(* IEC 61131-3 sources: LPWCC/src, 9 files *)

(* ---- GVL.st ---- *)
VAR_GLOBAL
	IX0_0 AT %IX0.0:BOOL;
	IX0_1 AT %IX0.1:BOOL;
	IX0_2 AT %IX0.2: BOOL;
	IX0_3 AT %IX0.3: BOOL;
	IX0_4 AT %IX0.4: BOOL;
	IX0_5 AT %IX0.5: BOOL;
	IX0_6 AT %IX0.6: BOOL;
	IX0_7 AT %IX0.7: BOOL;
	IX0_8 AT %IX0.8: BOOL;

	IW6 AT %IW6:WORD;
	IW7 AT %IW7:WORD;
	IW8 AT %IW8:WORD;
	IW9 AT %IW9:WORD;
	IW10 AT %IW10:WORD;
	IW11 AT %IW11:WORD;
	IW12 AT %IW12:WORD;
	IW13 AT %IW13:WORD;

	QX0_4 AT %QX0.4:BOOL;
	QX0_5 AT %QX0.5:BOOL;
	QX0_6 AT %QX0.6:BOOL;
	QX0_7 AT %QX0.7:BOOL;
	QX1_0 AT %QX1.0:BOOL;
	QX1_1 AT %QX1.1:BOOL;
	QX3_0 AT %QX3.0:BOOL;
	QX3_1 AT %QX3.1:BOOL;
	QX3_2 AT %QX3.2:BOOL;
	QX3_3 AT %QX3.3:BOOL;
	QX3_4 AT %QX3.4:BOOL;
	QX3_5 AT %QX3.5:BOOL;
	QX3_6 AT %QX3.6:BOOL;
	QX3_7 AT %QX3.7:BOOL;
	QX4_0 AT %QX4.0:BOOL;
	QX4_1 AT %QX4.1:BOOL;
	QX4_2 AT %QX4.2:BOOL;
	QX4_3 AT %QX4.3:BOOL;
	QX4_4 AT %QX4.4:BOOL;
	QX4_5 AT %QX4.5:BOOL;
	QX4_6 AT %QX4.6:BOOL;
	QX4_7 AT %QX4.7:BOOL;
	QX5_0 AT %QX5.0:BOOL;
	QX5_1 AT %QX5.1:BOOL;
	QX5_2 AT %QX5.2:BOOL;
	QX5_3 AT %QX5.3:BOOL;
	QX5_5 AT %QX5.5:BOOL;
	QW7 AT %QW7:WORD;
	QW8 AT %QW8:WORD;
	QW9 AT %QW9:WORD;
	QW10 AT %QW10:WORD;

	ExtRestart_State:BOOL;

	TON0_M_State:BOOL;
	TON1_M_State:BOOL;
	TON2_M_State:BOOL;
	TON3_M_State:BOOL;
	TON0_A_State:BOOL;
	TON1_A_State:BOOL;
	TON2_A_State:BOOL;
	TON3_A_State:BOOL;
	TON4_A_State:BOOL;
	TON5_A_State:BOOL;
	TON6_A_State:BOOL;
	TON7_A_State:BOOL;
	TON7_1_A_State:BOOL;
	TON7_2_A_State:BOOL;
	TON8_A_State:BOOL;
	TON8_1_A_State:BOOL;
	TON8_2_A_State:BOOL;
	TON9_A_State:BOOL;
	TON10_A_State:BOOL;
	TON11_A_State:BOOL;
	TON11_1_A_State:BOOL;
	TON12_A_State:BOOL;
	TON12_1_A_State:BOOL;
	TON13_State:BOOL;
	TON14_State:BOOL;
	TON15_State:BOOL;
	TON16_Emergency_stop:BOOL;
	TON17_State:BOOL;
	TON17_SW:BOOL;
	TON18_State:BOOL;
	TON18_SW:BOOL;
	TON19_State:BOOL;
	TON20_Emergency_stop:BOOL;
	TON21_A_State:BOOL;
	TON22_A_State:BOOL;

	CAN_SET_ArcOn:BOOL;
	CAN_SET_RobotReady:BOOL;
	CAN_SET_OperMode_0:BOOL;
	CAN_SET_OperMode_1:BOOL;
	CAN_SET_OperMode_2:BOOL;
	CAN_SET_AnalogSwap:BOOL;
	CAN_SET_ProtocolMode:BOOL;
	CAN_SET_GasTest:BOOL;
	CAN_SET_WireInching:BOOL;
	CAN_SET_WireRetract:BOOL;
	CAN_SET_SourceErrReset:BOOL;
	CAN_SET_TouchSensing:BOOL;
	CAN_SET_BlowTrough:BOOL;
	CAN_SET_JOB_0:BOOL;
	CAN_SET_JOB_1:BOOL;
	CAN_SET_JOB_2:BOOL;
	CAN_SET_JOB_3:BOOL;
	CAN_SET_JOB_4:BOOL;
	CAN_SET_JOB_5:BOOL;
	CAN_SET_JOB_6:BOOL;
	CAN_SET_JOB_7:BOOL;
	CAN_SET_WeldSim:BOOL;
	CAN_SET_AnalogSetDis_0:BOOL;
	CAN_SET_AnalogSetDis_1:BOOL;
	CAN_SET_AnalogSetDis_2:BOOL;
	CAN_SET_AnalogSetDis_3:BOOL;
	CAN_SET_AnalogSetDis_4:BOOL;
	CAN_SET_AnalogSetDis_5:BOOL;
	CAN_SET_DC_AC_Disable:BOOL;
	CAN_SET_PLS_Disable:BOOL;
	CAN_SET_DC_AC:BOOL;
	CAN_SET_PLS:BOOL;
	CAN_SET_PilotArc:BOOL;

	CAN_SET_WeldCurrent:UINT;
	CAN_SET_WireHighSpd:UINT;
	CAN_SET_PLS_Ratio:UINT;
	CAN_SET_WireLowSpd:UINT;
	CAN_SET_PlasmaGasFlow:UINT;
	CAN_SET_ShieldGasFlow:UINT;

	CAN_GET_CurrFlow:BOOL;
	CAN_GET_ProcActive:BOOL;
	CAN_GET_MainCurrent:BOOL;
	CAN_GET_CollisProtect:BOOL;
	CAN_GET_PowSourReady:BOOL;
	CAN_GET_Commun_Ready:BOOL;
	CAN_GET_ErrNumber_0:BOOL;
	CAN_GET_ErrNumber_1:BOOL;
	CAN_GET_ErrNumber_2:BOOL;
	CAN_GET_ErrNumber_3:BOOL;
	CAN_GET_ErrNumber_4:BOOL;
	CAN_GET_ErrNumber_5:BOOL;
	CAN_GET_ErrNumber_6:BOOL;
	CAN_GET_ErrNumber_7:BOOL;
	CAN_GET_PLS_Sync:BOOL;
	CAN_GET_PilotArc:BOOL;
	CAN_GET_StikingRem:BOOL;
	CAN_GET_WireAvailale:BOOL;

	CAN_GET_WeldVoltage:UINT;
	CAN_GET_WeldCurrent:UINT;
	CAN_GET_MotorCurrent:UINT;
	CAN_GET_WireFeedSPD:UINT;
	CAN_GET_PlasmaGasFlw:UINT;
	CAN_GET_ShieldGasFlw:UINT;

	MW110 AT %MW110:WORD;
	MW112 AT %MW112:WORD;
	MW114 AT %MW114:WORD;
	MW116 AT %MW116:WORD;
	MW118 AT %MW118:WORD;
	MW120 AT %MW120:WORD;
	MW122 AT %MW122:WORD;
	MW124 AT %MW124:WORD;
	MW126 AT %MW126:WORD;
	MW128 AT %MW128:WORD;

	TON0_FESTO:TON;
	TON0_FESTO_STATE:BOOL;
	TON0_FESTO_SW:BOOL;
	TON1_FESTO:TON;
	TON1_FESTO_STATE:BOOL;
	TON1_FESTO_SW:BOOL;
END_VAR

VAR_GLOBAL RETAIN
	MW0 AT %MW0:WORD;
	MW2 AT %MW2:WORD;
	MW4 AT %MW4:WORD;
	MW6 AT %MW6:WORD;
	MW8 AT %MW8:WORD;
	MW10 AT %MW10:WORD;
	MW12 AT %MW12:WORD;
	MW14 AT %MW14:WORD;
	MW16 AT %MW16:WORD;
	MW18 AT %MW18:WORD;
	MW20 AT %MW20:WORD;
	MW22 AT %MW22:WORD;
	MW24 AT %MW24:WORD;
	MW26 AT %MW26:WORD;
	MW28 AT %MW28:WORD;
	MW30 AT %MW30:WORD;
	MW32 AT %MW32:WORD;
	MW34 AT %MW34:WORD;
	MW36 AT %MW36:WORD;
	MW38 AT %MW38:WORD;
	MW40 AT %MW40:WORD;
	MW44 AT %MW44:WORD;
	MW42 AT %MW42:WORD;
	MW46 AT %MW46:WORD;
	MW48 AT %MW48:WORD;
	MW50 AT %MW50:WORD;
	MW52 AT %MW52:WORD;
	MW54 AT %MW54:WORD;
	MW56 AT %MW56:WORD;
	MW58 AT %MW58:WORD;
	MW60 AT %MW60:WORD;
	MW62 AT %MW62:WORD;
	MW64 AT %MW64:WORD;
	MW66 AT %MW66:WORD;
	MW68 AT %MW68:WORD;
	MW70 AT %MW70:WORD;
	MW72 AT %MW72:WORD;
	MW74 AT %MW74:WORD;
	MW76 AT %MW76:WORD;
	MW78 AT %MW78:WORD;
	MW80 AT %MW80:WORD;
	MW82 AT %MW82:WORD;
	MW84 AT %MW84:WORD;
	MW86 AT %MW86:WORD;
	MW88 AT %MW88:WORD;
	MW90 AT %MW90:WORD;
	MW92 AT %MW92:WORD;
	MW94 AT %MW94:WORD;
	MW96 AT %MW96:WORD;
	MW98 AT %MW98:WORD;
	MW100 AT %MW100:WORD;
	MW102 AT %MW102:WORD;
	MW104 AT %MW104:WORD;

	MW130 AT %MW130:WORD;
	MW132 AT %MW132:WORD;
	MW134 AT %MW134:WORD;
	MW136 AT %MW136:WORD;
	MW138 AT %MW138:WORD;
	MW140 AT %MW140:WORD;

	MD222 AT %MD222:DWORD;
	MD232 AT %MD232:DWORD;
	MD254 AT %MD254:DWORD;
	MD304 AT %MD304:DWORD;

END_VAR

(* ---- Alarms_auto.st ---- *)
VAR
	TON13: TON;
	TON14: TON;
	TON15: TON;
	TON16: TON;
END_VAR

//Затримка аналізу аварій
TON13(IN:= MW34.10, PT:= WORD_TO_TIME(MW96), Q=> TON13_State);
//Затримка аналізу чергової дуги
TON14(IN:= TON1_A_State, PT:= WORD_TO_TIME(MW60), Q=> TON14_State);
//Затримка аналізу основної дуги
TON15(IN:= (MW34.2 AND NOT(MW34.1) AND QX5_5) OR (MW34.1 AND CAN_SET_ArcOn) OR (MW34.9 AND QX5_3), PT:= WORD_TO_TIME(MW64), Q=> TON15_State);
//Аларми
IF TON13_State THEN
	IF IX0_0 THEN MW100:= 1; MW8.1:= TRUE; END_IF //Аларм по грибку
	IF MW18.12 AND IX0_8 THEN MW100:= 2; MW8.1:= TRUE; END_IF //Аларм по аварії лазера
	IF MW18.13 AND MW34.4 AND NOT(IX0_4) THEN MW100:= 3; MW8.1:= TRUE; END_IF //Аларм по неготовності робота
	IF MW18.14 AND MW34.4 AND IX0_6 THEN MW100:= 4; MW8.1:= TRUE; END_IF //Аларм по аварії робота
	IF MW8.6 AND IW6 < MW80 THEN MW100:= 5; MW8.1:= TRUE; END_IF //Аларм по низькому тиску газу зварювання
	IF MW8.7 AND IW7 < MW82 THEN MW100:= 6; MW8.1:= TRUE; END_IF //Аларм по низькому тиску газу різання
	IF MW8.8 AND IW8 < MW84 THEN MW100:= 7; MW8.1:= TRUE; END_IF //Аларм по низьких витратах газу зварювання
	IF MW8.9 AND IW9 < MW86 THEN MW100:= 8; MW8.1:= TRUE; END_IF //Аларм по низьких витратах газу різання
END_IF
IF MW8.12 AND MW18.8 AND TON13_State AND QX5_5 AND IW12 < MW92 THEN MW100:= 9; MW8.1:= TRUE; END_IF //Аларм по низькому струму різання
IF MW8.13 AND MW18.8 AND TON13_State AND QX5_5 AND IW13 < MW94 THEN MW100:= 10; MW8.1:= TRUE; END_IF //Аларм по низькій напрузі різання
IF MW8.10 AND MW18.8 AND TON13_State AND (CAN_SET_ArcOn OR CAN_SET_PilotArc) AND CAN_GET_WeldCurrent < MW88 THEN MW100:= 11; MW8.1:= TRUE; END_IF //Аларм низькому струму звар
IF MW8.11 AND MW18.8 AND TON13_State AND (CAN_SET_ArcOn OR CAN_SET_PilotArc) AND CAN_GET_WeldVoltage < MW90 THEN MW100:= 12; MW8.1:= TRUE; END_IF //Аларм по низькій напрузі звар
//Контроль на обрив чергової дуги
IF TON14_State AND TON13_State AND MW18.10 AND (CAN_SET_ArcOn OR CAN_SET_PilotArc) AND NOT(MW18.7) THEN MW100:= 13; MW8.1:= TRUE; END_IF
//Контроль на обрив основної дуги
IF TON15_State AND TON13_State AND MW18.11 AND NOT(MW18.8) THEN MW100:= 14; MW8.1:= TRUE; END_IF
//Скидання готовності при виникненні помилки
IF MW8.1 THEN MW8.2:= FALSE; END_IF
//Готовність в автоматі
IF NOT(MW8.1) AND NOT(IX0_0) AND ((MW34.4 AND ((MW18.13 AND IX0_4) OR NOT(MW18.13)) AND ((MW18.14 AND NOT(IX0_6)) OR NOT(MW18.14))) OR NOT(MW34.4)) AND ((MW18.12 AND MW34.00 AND NOT(IX0_8)) OR NOT(MW18.12) OR NOT(MW34.00)) AND ((MW8.6 AND IW6 >= MW80) OR NOT(MW8.6)) AND ((MW8.7 AND IW7 >= MW82) OR NOT(MW8.7)) THEN
	MW8.2:= TRUE; ELSE MW8.2:= FALSE; END_IF
//Затримка аварійного вимкнення
TON16(IN:= MW8.1, PT:= WORD_TO_TIME(MW98), Q=> TON16_Emergency_stop);
//Скидання аларму
IF MW8.0 THEN MW100:= 0; MW8.1:= FALSE; END_IF
QX4_4:= MW8.2; //Видача готовності шафи керування на робот

(* ---- Alarms_manual.st ---- *)
VAR
	TON13: TON;
	TON14: TON;
	TON15: TON;
	TON16: TON;
	TON19: TON;
	TON20: TON;
END_VAR

//Затримка аналізу аварій
TON19(IN:= MW0.7 OR MW0.9 OR MW0.10 OR MW0.11, PT:= WORD_TO_TIME(MW96), Q=> TON19_State);
//Аларми загальні
IF TON19_State THEN
	IF IX0_0 THEN MW100:= 1; MW8.1:= TRUE; END_IF //Аларм по грибку
	IF MW18.12 AND MW0.7 AND IX0_8 THEN MW100:= 2; MW8.1:= TRUE; END_IF //Аларм по аварії лазера
	IF MW8.6 AND IW6 < MW80 THEN MW100:= 5; MW8.1:= TRUE; END_IF //Аларм по низькому тиску газу зварювання
	IF MW8.7 AND IW7 < MW82 THEN MW100:= 6; MW8.1:= TRUE; END_IF //Аларм по низькому тиску газу різання
	IF MW8.8 AND IW8 < MW84 THEN MW100:= 7; MW8.1:= TRUE; END_IF //Аларм по низьких витратах газу зварювання
	IF MW8.9 AND IW9 < MW86 THEN MW100:= 8; MW8.1:= TRUE; END_IF //Аларм по низьких витратах газу різання
END_IF
IF MW8.12 AND MW18.8 AND TON19_State AND MW0.9 AND IW12 < MW92 THEN MW100:= 9; MW8.1:= TRUE; END_IF //Аларм по низькому струму різання
IF MW8.13 AND MW18.8 AND TON19_State AND MW0.9 AND IW13 < MW94 THEN MW100:= 10; MW8.1:= TRUE; END_IF //Аларм по низькій напрузі різання
IF MW8.10 AND MW18.8 AND TON19_State AND (MW0.10 OR MW0.11) AND CAN_GET_WeldCurrent < MW88 THEN MW100:= 11; MW8.1:= TRUE; END_IF //Аларм низькому струму звар
IF MW8.11 AND MW18.8 AND TON19_State AND (MW0.10 OR MW0.11) AND CAN_GET_WeldVoltage < MW90 THEN MW100:= 12; MW8.1:= TRUE; END_IF //Аларм по низькій напрузі звар
//Готовність лазера
IF NOT(MW8.1) AND NOT(IX0_0) AND ((MW18.12 AND NOT(IX0_8)) OR NOT(MW18.12)) AND ((MW8.6 AND IW6 >= MW80) OR NOT(MW8.6)) AND ((MW8.7 AND IW7 >= MW82) OR NOT(MW8.7)) THEN
	MW8.3:= TRUE; ELSE MW8.3:= FALSE; END_IF
//Готовність різання та зварювання + зварювання MIG
IF NOT(MW8.1) AND NOT(IX0_0) AND ((MW8.6 AND IW6 >= MW80) OR NOT(MW8.6)) AND ((MW8.7 AND IW7 >= MW82) OR NOT(MW8.7)) THEN
	MW8.4:= TRUE; MW8.5:= TRUE; MW8.15:= TRUE; ELSE MW8.4:= FALSE; MW8.5:= FALSE; MW8.15:= FALSE; END_IF
//Скидання готовностей при виникненні помилки
IF MW8.1 THEN MW8.3:= FALSE; MW8.4:= FALSE; MW8.5:= FALSE; MW8.15:= FALSE; END_IF
//Затримка аварійного вимкнення
TON20(IN:= MW8.1, PT:= WORD_TO_TIME(MW98), Q=> TON20_Emergency_stop);
//Скидання аларму
IF MW8.0 THEN MW100:= 0; MW8.1:= FALSE; END_IF
//Видача готовності шафи керування на робот
IF MW8.3 OR MW8.4 OR MW8.5 OR MW8.15 THEN QX4_4:= TRUE; ELSE QX4_4:= FALSE; END_IF

(* ---- Auto.st ---- *)
VAR
	TON1: TON;
	TON4: TON;
	TON2: TON;
	TON0: TON;
	TON7: TON;
	TON8: TON;
	TON7_1: TON;
	TON8_1: TON;
	TON7_2: TON;
	TON8_2: TON;
	TON6: TON;
	TON9: TON;
	TON10: TON;
	TON11: TON;
	TON12: TON;
	TON11_1: TON;
	TON12_1: TON;
	TON17: TON;
	TON18: TON;
	TON21: TON;
	TON22: TON;
END_VAR

//Індикація процесу на кнопці старт/стоп
TON17(IN:= NOT(TON17_SW), PT:= T#1S, Q=> TON17_State);
TON18(IN:= TON17_SW, PT:= T#1S, Q=> TON18_State);
IF TON17_State THEN TON17_SW:= TRUE; TON18_SW:= FALSE; END_IF
IF TON18_State THEN TON17_SW:= FALSE; TON18_SW:= TRUE; END_IF
IF MW34.10 THEN
	MW6:= 1;
ELSE
	IF MW34.7 THEN
		MW6:= 2;
	ELSE
		IF MW8.1 THEN
			IF TON17_SW THEN TON18_State:= FALSE; MW6:= 3; END_IF
			IF TON18_SW THEN TON17_State:= FALSE; MW6:= 0; END_IF
		ELSE
			MW6:= 0;
		END_IF
	END_IF
END_IF
//Застереження від повторного зовнішнього старту
IF NOT(IX0_5) THEN ExtRestart_State:= TRUE; END_IF

//Блок Are you sure/Stop
IF MW34.10 THEN MW34.6:= FALSE;
ELSE
	IF NOT(MW34.4) AND MW8.2 THEN MW34.6:= FALSE;
	ELSIF MW34.4 OR NOT(MW8.2) THEN MW34.6:= TRUE; END_IF
END_IF

//Трігери старт/стоп процесу
IF NOT(MW34.4) THEN
	IF TON16_Emergency_stop THEN MW34.10:= FALSE; END_IF
	IF MW34.8 THEN
		IF MW34.10 THEN MW34.10:= FALSE;
		ELSIF MW8.2 THEN MW34.5:= TRUE; END_IF
		MW34.8:= FALSE;
	END_IF
ELSE
	IF (MW34.10 AND MW34.8) OR NOT(IX0_5) OR TON16_Emergency_stop THEN MW34.10:= FALSE; MW34.8:= FALSE; END_IF
	IF IX0_5 AND ExtRestart_State AND MW8.2 THEN MW34.10:= TRUE; ExtRestart_State:=FALSE; END_IF
END_IF

//Цикл автоматичного режиму
TON1(IN:= MW34.10, PT:= WORD_TO_TIME(MW56), Q=> TON1_A_State); //T1
TON21(IN:= MW34.10, PT:= WORD_TO_TIME(MW134), Q=> TON21_A_State); //T13
//Конфігурація частотних виходів
FreqGen_0(EN_Enable:= TRUE, F_Enable:= TRUE, EN_Sync:= TRUE, F_Sync:= TRUE, Frequency:= MD254);
PWM_0(EN_Enable:= TRUE, F_Enable:= TRUE, EN_Sync:= TRUE, F_Sync:= TRUE,  Frequency:= MD222, Duty:= MW28);

//Задання попередніх параметрів зварювання до старту
CAN_SET_OperMode_1:= TRUE;
CAN_SET_OperMode_2:= TRUE;
CAN_SET_DC_AC := MW18.15;// Вибір режиму зварювання (AC або DC)
CAN_SET_WeldSim:= MW34.3;
CAN_SET_PlasmaGasFlow:= MW44;
CAN_SET_ShieldGasFlow:= MW46;

//START
IF MW34.10 THEN
	MW34.7:= TRUE; //In Process start
	//Керування подачею дроту та порошку
	TON7(IN:= MW2.13 AND (((MW34.1 OR MW34.2) AND MW18.8) OR (MW34.0 AND NOT(MW34.1) AND NOT(MW34.2))), PT:= WORD_TO_TIME(MW68), Q=> TON7_A_State);
	TON8(IN:= MW2.14 AND (((MW34.1 OR MW34.2) AND MW18.8) OR (MW34.0 AND NOT(MW34.1) AND NOT(MW34.2))), PT:= WORD_TO_TIME(MW70), Q=> TON8_A_State);
	IF TON7_A_State AND MW2.13 THEN QX5_0:= TRUE; END_IF
	IF TON8_A_State AND MW2.14 THEN QX5_1:= TRUE; END_IF
	IF NOT(MW2.13) THEN QX5_0:= FALSE; END_IF
	IF NOT(MW2.14) THEN QX5_1:= FALSE; END_IF
	//Керування газами
	IF MW2.1 THEN
		IF NOT(MW18.8) THEN QX3_1:= TRUE; END_IF
	ELSE QX3_1:= FALSE; END_IF
	IF MW2.6 THEN
		IF NOT(MW18.8) THEN QX3_6:= TRUE; END_IF
	ELSE QX3_6:= FALSE; END_IF
	QX3_0:= MW2.0; QX3_3:= MW2.3; QX3_4:= MW2.4; QX3_5:= MW2.5; QX4_1:= MW2.9; QX4_2:= MW2.10; QX4_3:= MW2.11;
	IF MW2.12 AND MW18.8 THEN MD254:= WORD_TO_DWORD(MW54); ELSE MD254:= 0; END_IF
	IF MW2.7 THEN
		IF MW18.8 THEN QX3_7:= TRUE; END_IF
	ELSE QX3_7:= FALSE; END_IF
	IF MW2.8 THEN
		IF MW18.8 THEN QX4_0:= TRUE; END_IF
	ELSE QX4_0:= FALSE; END_IF
	TON6(IN:= MW18.8, PT:= WORD_TO_TIME(MW66), Q=> TON6_A_State);
	IF TON6_A_State THEN QX3_1:= FALSE; QX3_6:= FALSE; END_IF
	//Керування лазером
	TON2(IN:= TON1_A_State AND MW34.0 AND ((NOT(MW34.1) AND NOT(MW34.2)) OR ((MW34.1 OR MW34.2) AND MW18.8)), PT:= WORD_TO_TIME(MW58), Q=> TON2_A_State);
	IF MW34.0 AND TON2_A_State THEN QW8:= MW36; END_IF
	TON0(IN:= MW34.0 AND TON2_A_State, PT:= T#20MS, Q=> TON0_A_State);
	IF TON0_A_State THEN QX1_0:= TRUE; QX1_1:= TRUE; MD222:= WORD_TO_DWORD(MW38); MW28:= MW40;
	ELSE QX1_0:= FALSE; QX1_1:= FALSE; MD222:=0; MW28:= 0; QW8:= 0; END_IF
	//Керування джерелом зварювання
	TON4(IN:= CAN_GET_PilotArc, PT:= WORD_TO_TIME(MW62), Q=> TON4_A_State);
	CAN_SET_RobotReady:= TRUE;
	IF MW34.1 THEN
		CAN_SET_WeldCurrent:= MW42;
		IF TON1_A_State THEN CAN_SET_PilotArc:= TRUE; END_IF
		IF TON4_A_State THEN CAN_SET_ArcOn:= TRUE; END_IF
	ELSE
		CAN_SET_ArcOn:= FALSE;
		CAN_SET_PilotArc:= FALSE;
		CAN_SET_WeldCurrent:= 0;
	END_IF
	//Керування джерелом різання
	IF MW34.2 THEN
		QW7:= MW48;
		IF TON1_A_State = TRUE THEN QX5_5:= TRUE; END_IF
	ELSE
		QX5_5:= FALSE;
		QW7:= 0;
	END_IF
	//Керування MIG джерелом
	IF MW34.9 THEN
		QW9:= MW138;
		QW10:= MW140;
		IF TON21_A_State = TRUE THEN QX5_3:= TRUE; END_IF
	ELSE
		QX5_3:= FALSE;
		QW9:= 0;
		QW10:= 0;
	END_IF
ELSE
//STOP
	//Керування джерелом зварювання
	CAN_SET_ArcOn:= FALSE;
	CAN_SET_PilotArc:= FALSE;
	CAN_SET_WeldCurrent:= 0;
	CAN_SET_RobotReady:= FALSE;
	//Керування джерелом різання
	QX5_5:= FALSE;
	QW7:= 0;
END_IF
//Керування подачею дроту та порошку
TON11(IN:= NOT(MW34.10), PT:= WORD_TO_TIME(MW76), Q=> TON11_A_State);
TON12(IN:= NOT(MW34.10), PT:= WORD_TO_TIME(MW78), Q=> TON12_A_State);
IF TON11_A_State THEN QX5_0:= FALSE; END_IF
IF TON12_A_State THEN QX5_1:= FALSE; END_IF
//Керування газами
TON10(IN:= NOT(MW34.10), PT:= WORD_TO_TIME(MW74), Q=> TON10_A_State);
IF TON10_A_State THEN
	QX3_0:= FALSE; QX3_1:= FALSE; QX3_3:= FALSE; QX3_4:= FALSE; QX3_5:= FALSE; QX3_6:= FALSE; QX3_7:= FALSE;
	QX4_0:= FALSE; QX4_1:= FALSE; QX4_2:= FALSE; QX4_3:= FALSE; MD254:= 0;
END_IF
//Керування лазером
TON9(IN:= NOT(MW34.10), PT:= WORD_TO_TIME(MW72), Q=> TON9_A_State);
IF TON9_A_State THEN QX1_0:= FALSE; QX1_1:= FALSE; MD222:=0; MW28:= 0; QW8:= 0; END_IF
//Керування MIG джерелом
TON22(IN:= NOT(MW34.10), PT:= WORD_TO_TIME(MW136), Q=> TON22_A_State); //T14
IF TON22_A_State THEN QX5_3:= FALSE; QW9:= 0; QW10:= 0; END_IF
//In Process stop
IF TON9_A_State AND TON10_A_State AND TON11_A_State AND TON12_A_State THEN MW34.7:= FALSE; END_IF
QX4_6:= MW34.7; //Видача In progress на робот

(* ---- Default.st ---- *)
VAR
	I: INT;
END_VAR

MW34.10:= FALSE;
MW0.7:= FALSE;
MW0.9:= FALSE;
MW0.10:= FALSE;
MW0.11:= FALSE;
MW4.1:= FALSE;
MW4.2:= FALSE;
MW4.3:= FALSE;
MW4.4:= FALSE;
MW4.5:= FALSE;
MW4.7:= FALSE;
MW4.8:= FALSE;
MW4.9:= FALSE;
MW4.10:= FALSE;
MW4.11:= FALSE;
MW4.12:= FALSE;
MW4.13:= FALSE;
MW4.14:= FALSE;
MW18.1:= FALSE;
MW18.2:= FALSE;
MD254:= 0;
MD304:= 0;
QX3_0:= FALSE;
QX3_1:= FALSE;
QX3_2:= FALSE;
QX3_3:= FALSE;
QX3_4:= FALSE;
QX3_5:= FALSE;
QX3_6:= FALSE;
QX3_7:= FALSE;
QX4_0:= FALSE;
QX4_1:= FALSE;
QX4_2:= FALSE;
QX4_3:= FALSE;
QX1_0:= FALSE;
QX1_1:= FALSE;
QX5_0:= FALSE;
QX5_1:= FALSE;
MD222:=0;
MW28:= 0;
QW8:= 0;
CAN_SET_ArcOn:= FALSE;
CAN_SET_PilotArc:= FALSE;
CAN_SET_WeldCurrent:= 0;
CAN_SET_RobotReady:= FALSE;
QX5_5:= FALSE;
QW7:= 0;
QX5_3:= FALSE;
QW9:= 0;
QW10:= 0;
//Конфігурація частотних виходів
FreqGen_0(EN_Enable:= TRUE, F_Enable:= TRUE, EN_Sync:= TRUE, F_Sync:= TRUE, Frequency:= MD254);
FreqGen_1(EN_Enable:= TRUE, F_Enable:= TRUE, EN_Sync:= TRUE, F_Sync:= TRUE, Frequency:= MD304);
PWM_0(EN_Enable:= TRUE, F_Enable:= TRUE, EN_Sync:= TRUE, F_Sync:= TRUE,  Frequency:= MD222, Duty:= MW28);

(* ---- LaserCut_focus.st ---- *)
VAR
	TON3_State: BOOL;
	TON2_State: BOOL;
	TON1_State: BOOL;
	TON0_State: BOOL;
	TON3: TON;
	TON2: TON;
	TON1: TON;
	TON0: TON;
END_VAR

//Керування двигуном позиціонування лазерної головки (в меню опції)
FreqGen_1(EN_Enable:= TRUE, F_Enable:= TRUE, EN_Sync:= TRUE, F_Sync:= TRUE, Frequency:= MD304);
TON0(IN:= MW34.11, PT:= T#1MS, Q=> TON0_State); //Задання напрямку 1
TON3(IN:= MW34.12, PT:= T#1MS, Q=> TON3_State); //Задання напрямку 2
TON1(IN:= TON0_State OR TON3_State, PT:= T#1MS, Q=> TON1_State); //Старт частоти
TON2(IN:= NOT(MW34.11) AND NOT(MW34.12), PT:= T#1MS, Q=> TON2_State); //Взведення ENA (стоп)
IF MW34.11 THEN
	MW34.12:= FALSE; QX0_7:= FALSE;
	IF TON0_State THEN QX0_6:= FALSE; END_IF
	IF TON1_State THEN MD304:= WORD_TO_DWORD(MW104)*10; END_IF
END_IF
IF MW34.12 THEN
	MW34.11:= FALSE; QX0_7:= FALSE;
	IF TON3_State THEN QX0_6:= TRUE; END_IF
	IF TON1_State THEN MD304:= WORD_TO_DWORD(MW104)*10; END_IF
END_IF
IF NOT(MW34.11) AND NOT(MW34.12) THEN
	MD304:= 0;
	IF TON2_State THEN QX0_7:= TRUE; END_IF
END_IF

(* ---- Main.st ---- *)
VAR
	RTRIG1: R_TRIG;
END_VAR

QX4_7:= TRUE; //Подача сигналу "Керування від ЛПЗР" на Schneider-робота
IF MW0.5 THEN  Alarms_manual(); ELSE Alarms_auto(); END_IF //Аларми
Measure();
RTRIG1(CLK:= NOT(MW0.5));
IF IX0_0 OR RTRIG1.Q THEN Default(); END_IF //Скидання до дефолту
IF MW0.5 THEN  Manual(); LaserCut_focus(); ELSE Auto(); END_IF //Ручний + laser focus / Автоматичний

(* ---- Manual.st ---- *)
VAR
	WORD_AS_BIT_1: WORD_AS_BIT;
	TON0: TON;
	TON1: TON;
	TON2: TON;
	TON3: TON;
	TON17: TON;
	TON18: TON;
END_VAR

//Індикація мигання надпису ALARM
TON17(IN:= NOT(TON17_SW), PT:= T#1MS, Q=> TON17_State);
TON18(IN:= TON17_SW, PT:= T#1S, Q=> TON18_State);
IF TON17_State THEN TON17_SW:= TRUE; TON18_SW:= FALSE; END_IF
IF TON18_State THEN TON17_SW:= FALSE; TON18_SW:= TRUE; END_IF
IF MW8.1 THEN
	IF TON17_SW THEN TON18_State:= FALSE; MW102:= 1; END_IF
	IF TON18_SW THEN TON17_State:= FALSE; MW102:= 0; END_IF
END_IF

//Керування газами
WORD_AS_BIT_1( W:= MW4,B01=> QX3_0, B02=> QX3_1, B04=> QX3_3, B05=> QX3_4, B07=> QX3_5, B08=> QX3_6, B09=> QX3_7, B10=> QX4_0, B11=> QX4_1, B12=> QX4_2, B13=> QX4_3);
//Частотний клапан FESTO
IF MW4.14 THEN MD232:= WORD_TO_DWORD(MW32); ELSE MD232:= 0; END_IF
FreqGen_0(EN_Enable:= TRUE, F_Enable:= TRUE, EN_Sync:= TRUE, F_Sync:= TRUE, Frequency:= MD232);
//Керування двигуном подачі дроту
QX5_0:= MW18.1;
//Керування двигуном подачі порошку
QX5_1:= MW18.2;
//Керування лазером
IF MW0.7 OR (MW0.6 AND MW8.3) THEN MW0.8:= FALSE; ELSE MW0.8:= TRUE; END_IF
IF MW0.6 THEN
	QW8:= MW20;
ELSE
	QW8:= 0;
END_IF
IF MW0.7 AND MW8.3 THEN
	QX1_0:= TRUE;
	QX1_1:= TRUE;
	MD222:= WORD_TO_DWORD(MW22);
	MW28:= MW26;
ELSIF NOT(MW0.7) OR TON20_Emergency_stop THEN
	MW0.7:= FALSE;
	QX1_0:= FALSE;
	QX1_1:= FALSE;
	MD222:= 0;
	MW28:= 0;
END_IF
PWM_0(
	EN_Enable:= TRUE,
	F_Enable:= TRUE,
	EN_Sync:= TRUE,
	F_Sync:= TRUE,
	Frequency:= MD222,
	Duty:= MW28);

//Керування джерелом різання
IF MW0.9 OR (MW0.13 AND MW8.4) THEN MW0.15:= FALSE; ELSE MW0.15:= TRUE; END_IF
IF MW0.13 THEN
	QW7:= MW16;
ELSE
	QW7:= 0;
END_IF
IF MW0.9 AND MW8.4 THEN
	QX5_5:= TRUE;
ELSIF NOT(MW0.9) OR TON20_Emergency_stop THEN
	MW0.9:= FALSE;
	QX5_5:= FALSE;
END_IF

//Керування джерелом MIG
IF MW34.15 OR (MW34.13 AND MW8.15) THEN MW34.14:= FALSE; ELSE MW34.14:= TRUE; END_IF
IF MW34.13 THEN
	QW9:= MW130;
	QW10:= MW132;
ELSE
	QW9:= 0;
	QW10:= 0;
END_IF
IF MW34.15 AND MW8.15 THEN
	QX5_3:= TRUE;
ELSIF NOT(MW34.15) OR TON20_Emergency_stop THEN
	MW34.15:= FALSE;
	QX5_3:= FALSE;
END_IF

//Керування джерелом зварювання
IF MW0.10 OR MW0.11 OR (MW0.12 AND MW8.5) THEN MW0.14:= FALSE; ELSE MW0.14:= TRUE; END_IF
IF MW0.10 OR MW0.11 THEN MW2.2:= TRUE; ELSE MW2.2:= FALSE; END_IF
CAN_SET_WeldSim:= MW0.0;
CAN_SET_PlasmaGasFlow:= MW24;
CAN_SET_ShieldGasFlow:= MW30;
CAN_SET_OperMode_1:= TRUE;
CAN_SET_OperMode_2:= TRUE;
CAN_SET_DC_AC := MW18.15;// Вибір режиму зварювання (AC або DC)
IF MW0.12 THEN
	CAN_SET_RobotReady:= TRUE;
	CAN_SET_WeldCurrent:= MW12;
ELSE
	CAN_SET_RobotReady:= FALSE;
	CAN_SET_WeldCurrent:= 0;
END_IF
IF MW0.10 AND MW8.5 THEN
	CAN_SET_PilotArc:= TRUE;
	IF MW0.11 AND MW8.5 THEN
		CAN_SET_ArcOn:= TRUE;
	ELSIF NOT(MW0.11) OR TON20_Emergency_stop THEN
		MW0.11:= FALSE;
		CAN_SET_ArcOn:= FALSE;
	END_IF
ELSIF NOT(MW0.10) OR TON20_Emergency_stop THEN
	MW0.10:= FALSE;
	MW0.11:= FALSE;
	CAN_SET_PilotArc:= FALSE;
	CAN_SET_ArcOn:= FALSE;
	MW0.11:= FALSE;
END_IF
//Блок переходу в автомат та видача IN PROGRESS в ручному режимі
IF CAN_SET_ArcOn OR CAN_SET_PilotArc OR QX5_5 OR QX5_3 OR QX1_0 OR QX1_1 THEN MW8.14:= TRUE; QX4_6:= TRUE; ELSE MW8.14:= FALSE; QX4_6:= FALSE; END_IF

(* ---- Measure.st ---- *)
//Дискретні сигнали
MW18.3:= IX0_0;
MW18.4:= IX0_8;
MW18.5:= IX0_4;
MW18.6:= IX0_6;
MW18.9:= IX0_5;
MW18.7:= CAN_GET_PilotArc;
IF QX5_5 AND (CAN_SET_ArcOn OR CAN_SET_PilotArc) THEN MW18.8:= IX0_2 AND CAN_GET_MainCurrent;
ELSIF QX5_3 AND (CAN_SET_ArcOn OR CAN_SET_PilotArc) THEN MW18.8:= IX0_3 AND CAN_GET_MainCurrent;
ELSIF CAN_SET_ArcOn OR CAN_SET_PilotArc THEN MW18.8:= CAN_GET_MainCurrent;
ELSIF QX5_5 THEN MW18.8:= IX0_2;
ELSIF QX5_3 THEN MW18.8:= IX0_3;
ELSIF NOT(IX0_2) AND NOT(CAN_GET_MainCurrent) AND NOT(IX0_3) THEN MW18.8:= FALSE; END_IF
QX4_5:= MW18.8; //Видача Main current на робот

//Аналогові входи
IF IW12 >= 4800 THEN //Cutting current
	MW114:= IW12;
ELSE
	MW114:= 4000;
END_IF
IF IW13 >= 4500 THEN //Cutting voltage
	MW116:= IW13;
ELSE
	MW116:= 4000;
END_IF
IF IW6 >= 4100 THEN //BP1 pl. wel.
	MW118:= IW6;
ELSE
	MW118:= 4000;
END_IF
IF IW7 >= 4100 THEN //BP2 pl. cut.
	MW120:= IW7;
ELSE
	MW120:= 4000;
END_IF
IF IW8 >= 4100 THEN //FT2 pl. wel.
	MW122:= IW8;
ELSE
	MW122:= 4000;
END_IF
IF IW9 >= 4100 THEN //FT7 pl. cut.
	MW124:= IW9;
ELSE
	MW124:= 4000;
END_IF

//Вимірювання струму зварювання Cebora
IF CAN_GET_WeldCurrent <= 655 THEN
	MW110:= 0;
ELSE
	MW110:= CAN_GET_WeldCurrent;
END_IF

//Вимірювання напруги зварювання Cebora
IF CAN_GET_WeldVoltage <= 5000 THEN
	MW112:= 0;
ELSE
	MW112:= CAN_GET_WeldVoltage;
END_IF

//Вимірювання Cebora plasma gas
IF CAN_GET_PlasmaGasFlw <= 655 THEN
	MW126:= 0;
ELSE
	MW126:= CAN_GET_PlasmaGasFlw;
END_IF

//Вимірювання Cebora shield gas
IF CAN_GET_ShieldGasFlw <= 220 THEN
	MW128:= 0;
ELSE
	MW128:= CAN_GET_ShieldGasFlw;
END_IF
